Fanuc KAREL source: RENAME_VAR.kl

PROGRAM T
%NOLOCKGROUP
VAR
 v0 : STRING[40]
 v1 : STRING[40]
 v2 : STRING[40]
 v3 : INTEGER
BEGIN
 RENAME_VAR(v0, v1, v2, v3)
END T
